// Mitsubishi GX Works2 project: z11   PLC: Q02/Q02H

PROGRAM MAIN
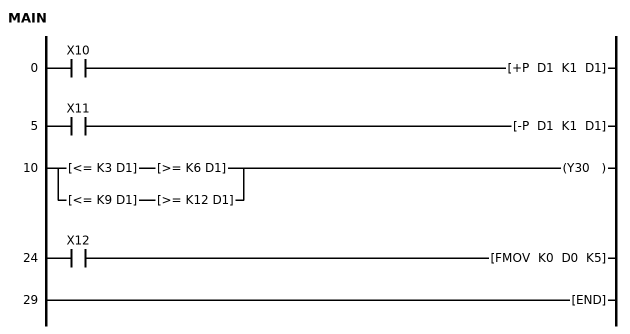
0     LD      X10
      +P      D1 K1 D1
5     LD      X11
      -P      D1 K1 D1
10    LD<=    K3 D1
      AND>=   K6 D1
      LD<=    K9 D1
      AND>=   K12 D1
      ORB
      OUT     Y30
24    LD      X12
      FMOV    K0 D0 K5
29    END
END_PROGRAM
